{attribute 'linkalways'} 
{attribute 'no_explicit_call' := 'This FB is a CLASS and must be accessed using methods or properties'}
{attribute 'enable_dynamic_creation'}
FUNCTION_BLOCK Node_F_VN_GetAt_TcVnRectangle_DINT EXTENDS VisionNode
VAR
    ipContainer : _ITcVnContainer;
    stElement : _TcVnRectangle_DINT;
    nIndex : _ULINT(0);
    hrPrev : _HRESULT(S_OK);
    hresult : _HRESULT(S_OK);
END_VAR

METHOD PUBLIC  Clone : I_Node
VAR
	pNode : POINTER TO Node_F_VN_GetAt_TcVnRectangle_DINT;
END_VAR
pNode := __NEW(Node_F_VN_GetAt_TcVnRectangle_DINT);
Clone := pNode^;
END_METHOD

METHOD FB_init : BOOL
VAR_INPUT
	bInitRetains : BOOL; // if TRUE, the retain variables are initialized (warm start / cold start)
	bInCopyCode : BOOL;  // if TRUE, the instance afterwards gets moved into the copy code (online change)
END_VAR
AddInput('ipContainer', ipContainer);
AddInput('nIndex', nIndex);
AddInput('hrPrev', hrPrev);
AddOutput('stElement', stElement);
AddOutput('hresult',hresult);
END_METHOD

METHOD PROTECTED OnExecute : HRESULT
hresult.Value := F_VN_GetAt_TcVnRectangle_DINT(
    ipContainer := ipContainer.Value,
    stElement := stElement.Value,
    nIndex := nIndex.Value,
    hrPrev:= hrPrev.Value);
END_METHOD

METHOD PUBLIC PreExecutionCheck
VAR_INPUT
	Check : I_PreExecutionChecks;
END_VAR
Check.IsTrue(ipContainer.IsValid, 'ipContainer must be a valid container');
Check.IsTrue(ipContainer.HasType(TC_GLOBAL_CONST_LIST.ContainerType_Vector_TcVnRectangle_DINT), 'ipContainer contains incorrect type');
END_METHOD

END_FUNCTION_BLOCK

(* stored: Version 1.1.0.1, ProductVersion 3.1.4024.13
   POU Node_F_VN_GetAt_TcVnRectangle_DINT: Id {9b0ab18f-b965-43fb-a1bf-c6294958d4e8}, SpecialFunc None
   Folder Constructor: Id {809852bf-87a9-4335-b79e-1cc076ae1598}
   Method Clone: Id {3a69a29b-069f-4192-a7b4-57e02e442cff}
   Method FB_init: Id {4577d2bd-1ced-4262-a1b4-e9f59cca8f19}
   Method OnExecute: Id {e20e3016-790e-474d-8332-251db6604826}
   Method PreExecutionCheck: Id {43cfb219-15e6-490a-89ac-1351854f3113} *)
